(* IEC 61131-3 sources: teller/JD_Teller_LC2_V11/Class/ETV0551_IOs, 1 file *)

(* ---- ETV0551_IOs.st ---- *)
(*!
<Class
	Name               = "ETV0551_IOs"
	Revision           = "1.10"
	RealtimeTask       = "false"
	CyclicTask         = "false"
	BackgroundTask     = "false"
	Sigmatek           = "true"
	OSInterface        = "false"
	HighPriority       = "false"
	Automatic          = "false"
	UpdateMode         = "Prescan"
	IconPath           = ".\Class\DigInOut.ICO"
	SharedCommandTable = "true"
	Objectsize         = "(426,120)"
	Comment            = "Class to access digital IOs on ETV0551 (8xDigIn, 8xDigOut)">
	<Channels>
	</Channels>
	<RevDoku>
		<Owner Company="Sigmatek" Author="RamAnd"/>
		<Dokumentation Revision="1.10" Date="06.12.2013" Author="LanSte" Company="Sigmatek" Description="Hardware class description file (lhd) updated."/>
		<Dokumentation Revision="1.4" Date="15.02.2012" Author="RamAnd" Company="Sigmatek" Description="Outputs are only written to hardware, if they have changed."/>
		<Dokumentation Revision="1.3" Date="27.10.2010" Author="RamAnd" Company="Sigmatek" Description="Added RtPostScan support"/>
		<Dokumentation Revision="1.2" Date="15.10.2010" Author="BleErn" Company="Sigmatek" Description="Content of corresponding LASAL Hardware Description file (.lhd) which is necessary for the hardware editor has been updated"/>
		<Dokumentation Revision="1.1" Date="13.07.2010" Author="BleErn" Company="Sigmatek" Description="Content of corresponding LASAL Hardware Description file (.lhd) which is necessary for the hardware editor has been corrected"/>
		<Dokumentation Revision="1.0" Date="01.03.2010" Author="RamAnd" Company="Sigmatek" Description="Initial Version"/>
	</RevDoku>
	<Network Name="ETV0551_IOs">
		<!-- List of Components in this network -->
		<Components>
			<Object
				Name       = "_base"
				Class      = "ETVEdge_DigIO_Base"
				Position   = "(218,120)"
				Visualized = "false"
				CyclicTime = "100 ms">
				<Channels>
					<Server Name="Input1"/>
					<Server Name="Input2"/>
					<Server Name="Input3"/>
					<Server Name="Input4"/>
					<Server Name="Input5"/>
					<Server Name="Input6"/>
					<Server Name="Input7"/>
					<Server Name="Input8"/>
					<Server Name="InputByte"/>
					<Server Name="Output1"/>
					<Server Name="Output2"/>
					<Server Name="Output3"/>
					<Server Name="Output4"/>
					<Server Name="Output5"/>
					<Server Name="Output6"/>
					<Server Name="Output7"/>
					<Server Name="Output8"/>
					<Server Name="OutputByte"/>
					<Server Name="State"/>
					<Client Name="To_HwControl"/>
				</Channels>
			</Object>
		</Components>
		<Comments>
		</Comments>
		<!-- List of Connections in this network -->
		<Connections>
			<Connection Source="this.State" Destination="_base.State" Vertices="(832,210),(660,210),"/>
			<Connection Source="this.Input1" Destination="_base.Input1" Vertices="(832,270),(660,270),"/>
			<Connection Source="this.Input2" Destination="_base.Input2" Vertices="(832,330),(660,330),"/>
			<Connection Source="this.Input3" Destination="_base.Input3" Vertices="(832,390),(660,390),"/>
			<Connection Source="this.Input4" Destination="_base.Input4" Vertices="(832,450),(660,450),"/>
			<Connection Source="this.Input5" Destination="_base.Input5" Vertices="(832,510),(660,510),"/>
			<Connection Source="this.Input6" Destination="_base.Input6" Vertices="(832,570),(660,570),"/>
			<Connection Source="this.Input7" Destination="_base.Input7" Vertices="(832,630),(660,630),"/>
			<Connection Source="this.Input8" Destination="_base.Input8" Vertices="(832,690),(660,690),"/>
			<Connection Source="this.Output1" Destination="_base.Output1" Vertices="(832,750),(660,750),"/>
			<Connection Source="this.Output2" Destination="_base.Output2" Vertices="(832,810),(660,810),"/>
			<Connection Source="this.Output3" Destination="_base.Output3" Vertices="(832,870),(660,870),"/>
			<Connection Source="this.Output4" Destination="_base.Output4" Vertices="(832,930),(660,930),"/>
			<Connection Source="this.Output5" Destination="_base.Output5" Vertices="(832,990),(660,990),"/>
			<Connection Source="this.Output6" Destination="_base.Output6" Vertices="(832,1050),(660,1050),"/>
			<Connection Source="this.Output7" Destination="_base.Output7" Vertices="(832,1110),(660,1110),"/>
			<Connection Source="this.Output8" Destination="_base.Output8" Vertices="(832,1170),(660,1170),"/>
			<Connection Source="this.InputByte" Destination="_base.InputByte" Vertices="(832,1230),(660,1230),"/>
			<Connection Source="this.OutputByte" Destination="_base.OutputByte" Vertices="(832,1290),(660,1290),"/>
			<Connection Source="_base.To_HwControl" Destination="this.To_HwControl" Vertices="(218,210),(38,210),"/>
		</Connections>
		<!-- Headerfiles -->
		<Options>
		</Options>
	</Network>
</Class>
*)
#pragma using ETVEdge_DigIO_Base

ETV0551_IOs : CLASS
: ETVEdge_DigIO_Base
  //Servers:
  //Clients:
  //Variables:
  //Functions:
  //Tables:
	FUNCTION @STD
		VAR_OUTPUT
			ret_code	: CONFSTATES;
		END_VAR;
	FUNCTION GLOBAL TAB @CT_;
END_CLASS;
